# EPICS substitutions: CS-RF-IOC-01/CS-RF-IOC-01App/Db/CS-RF-IOC-01.substitutions
################################################################################

file ../SR-RF-LN2-02.template
{
	pattern
	{
		device, port
	}
	{
		SR-RF-LN2-02, LN2
	}
}
